(* Logix 5000 project; controller R5_CSS vendor 1 type 14 code 74 rev 19.11; software revision 19.01; part 10 of 20 *)
(* tags used below, declared in another part *)
   CSS_SHUT_PALL : BOOL;
   AlarmMaster : DINT;
   AllowHeatersWhenEmpty : BOOL;
   AllowHeatersWhenEmpty_MaxMin : DINT;
   AllowHeatersWhenEmpty_ONS : BOOL;
   AllowHeatersWhenEmpty_SecRemaining : DINT;
   AllowHeatersWhenEmptyTON : TIMER;
   CSS_Heartbeat : BOOL;
   CSS_HeartbeatTmr : TIMER;
   CSS_HeartbeatToggle : BOOL;
   CSS_OK_TO_RUN : BOOL;   // PRU_RUN_DISABLE 0 = Cannot Run 1 = OK to Run
   CSS_OK_TO_RUN_TOF : TIMER;
   CSS_OK_TO_START : BOOL;   // PRU_START_DISABLE 0 = Cannot Start 1 = OK to Start
   CSS_OK_TO_START_TOF : TIMER;
   HART1 : HARTModuleDef;
   HeaterControl_IgnoreLevel : BOOL;
   HeaterControl_IgnoreLevel_ONS : BOOL;
   LC101 : LEVEL_CONTROL;   // QUENCH TOWER BASIN LIT
   LC205 : LEVEL_CONTROL;   // OVERHEAD CONDENSER BASIN LEVEL CONTROL
   LC205_START_SP : REAL;
   LC205_STOP_SP : REAL;
   LC303A : LEVEL_CONTROL;   // AQUEOUS PHASE OF PRIMARY SETTLER
   LC303B : LEVEL_CONTROL;   // INTERFACE LEVEL OF PRIMARY CONDENSER
   LC303C : LEVEL_CONTROL;   // DIFFERENCE BETWEEN INTERFACE AND AQUEOUS PHASE LT 303
   MV115B : ValveControl_TwoWay;
   MV301 : ValveControl_TwoWay;
   ONE_SHOT : BOOL[32];
   P101A : PUMP_CONTROL;
   P101A_OK : BOOL;
   P101B : PUMP_CONTROL;
   P101B_OK : BOOL;
   P205 : PUMP_CONTROL;   // OVERHEAD CONDENSER TRANSFER PUMP
   P205_QI_AUTO_OS : BOOL;
   P205_QI_MAN_OS : BOOL;
   P302A : PUMP_CONTROL;
   P302A_OK : BOOL;
   P302A_PumpOut : BOOL;
   P302B : PUMP_CONTROL;
   P302B_OK : BOOL;
   P302B_PumpOut : BOOL;
   P303A : PUMP_CONTROL;
   P303A_OK : BOOL;
   P303B : PUMP_CONTROL;
   P303B_OK : BOOL;
   PC407B : PRESSURE_CONTROL;   // POST HX LOW PRESSURE TRANSMITTER
   TC101A : TEMP_CONTROL;   // QUENCH BASIN TRANSFER BASIN A TEMPERATURE CONTROL
   TC101B : TEMP_CONTROL;   // QUENCH BASIN TRANSFER BASIN B TEMPERATURE CONTROL
   TC108 : TEMP_CONTROL;   // QUENCH TOWER EXIT GAS TEMPERATURE CONTROL
   TC112 : TEMP_CONTROL;   // Quench Water Cartridge Heater ProcessTemp
   TC313A : TEMP_CONTROL;   // PRIMARY COALESCER SEPARATOR TEMPERATURE CONTROL
   TC319 : TEMP_CONTROL;   // COALESCER OIL CHAMBER PROCESS TEMPERATURE CONTROL
   TestyBit : DINT;
   TMR_CRIT_FAULT : DINT;
   TMR_FAULT : DINT;
   UTL_Comms : DINT[3];
(* MainProgram, continued *)

ROUTINE LCV303C_COPY_CoalPriChamberInterfaceDiff   (* ladder *)
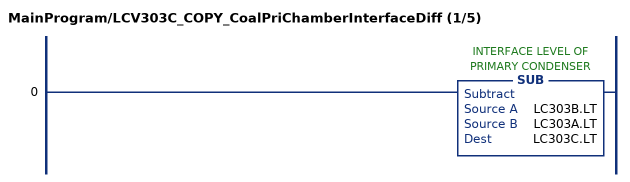
   0: SUB(LC303B.LT,LC303A.LT,LC303C.LT);
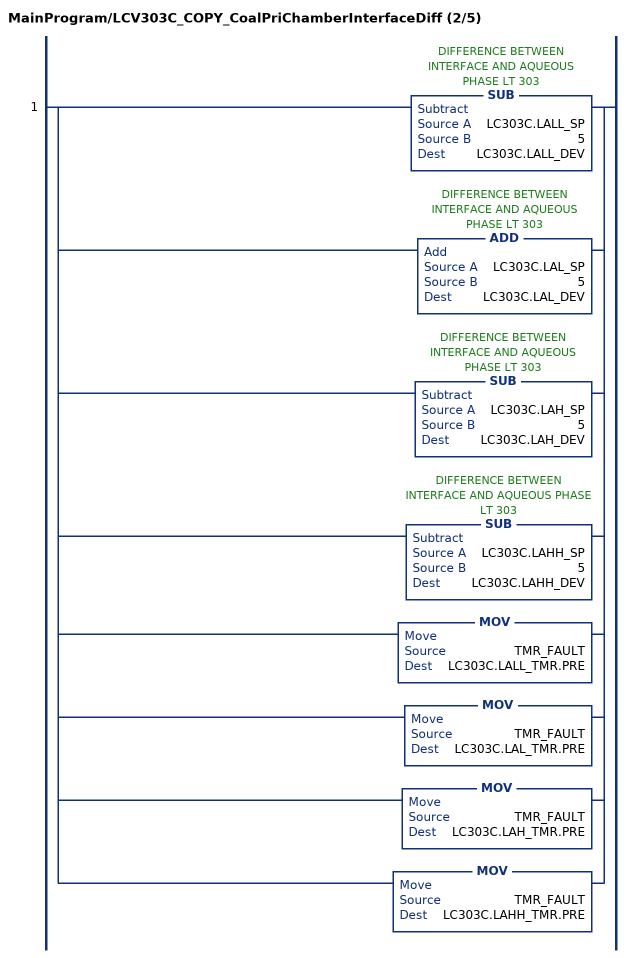
   1: [SUB(LC303C.LALL_SP,5,LC303C.LALL_DEV) ,ADD(LC303C.LAL_SP,5,LC303C.LAL_DEV) ,SUB(LC303C.LAH_SP,5,LC303C.LAH_DEV) ,SUB(LC303C.LAHH_SP,5,LC303C.LAHH_DEV) ,MOV(TMR_FAULT,LC303C.LALL_TMR.PRE) ,MOV(TMR_FAULT,LC303C.LAL_TMR.PRE) ,MOV(TMR_FAULT,LC303C.LAH_TMR.PRE) ,MOV(TMR_FAULT,LC303C.LAHH_TMR.PRE) ];
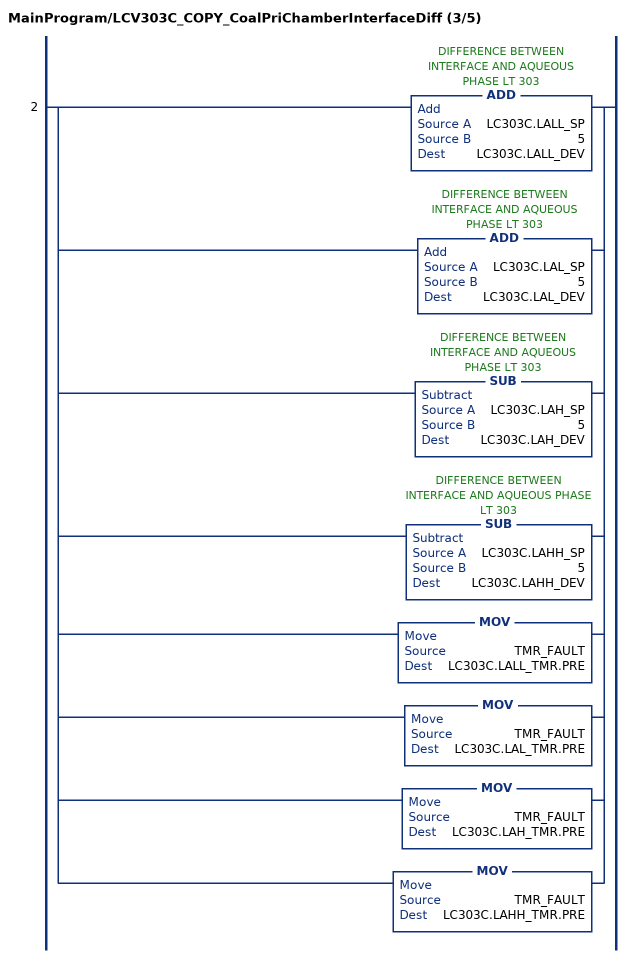
   2: [ADD(LC303C.LALL_SP,5,LC303C.LALL_DEV) ,ADD(LC303C.LAL_SP,5,LC303C.LAL_DEV) ,SUB(LC303C.LAH_SP,5,LC303C.LAH_DEV) ,SUB(LC303C.LAHH_SP,5,LC303C.LAHH_DEV) ,MOV(TMR_FAULT,LC303C.LALL_TMR.PRE) ,MOV(TMR_FAULT,LC303C.LAL_TMR.PRE) ,MOV(TMR_FAULT,LC303C.LAH_TMR.PRE) ,MOV(TMR_FAULT,LC303C.LAHH_TMR.PRE) ];
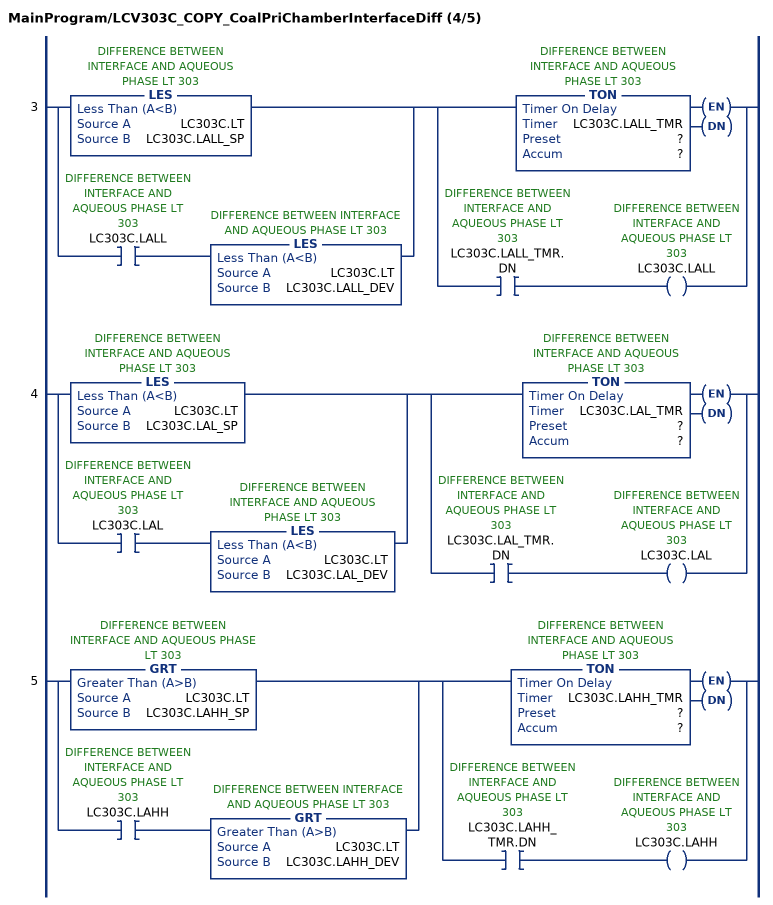
   3: [LES(LC303C.LT,LC303C.LALL_SP) ,XIC(LC303C.LALL) LES(LC303C.LT,LC303C.LALL_DEV) ][TON(LC303C.LALL_TMR,?,?) ,XIC(LC303C.LALL_TMR.DN) OTE(LC303C.LALL) ];
   4: [LES(LC303C.LT,LC303C.LAL_SP) ,XIC(LC303C.LAL) LES(LC303C.LT,LC303C.LAL_DEV) ][TON(LC303C.LAL_TMR,?,?) ,XIC(LC303C.LAL_TMR.DN) OTE(LC303C.LAL) ];
   5: [GRT(LC303C.LT,LC303C.LAHH_SP) ,XIC(LC303C.LAHH) GRT(LC303C.LT,LC303C.LAHH_DEV) ][TON(LC303C.LAHH_TMR,?,?) ,XIC(LC303C.LAHH_TMR.DN) OTE(LC303C.LAHH) ];
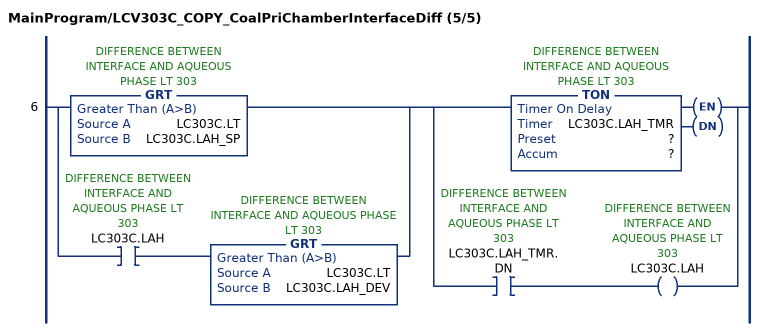
   6: [GRT(LC303C.LT,LC303C.LAH_SP) ,XIC(LC303C.LAH) GRT(LC303C.LT,LC303C.LAH_DEV) ][TON(LC303C.LAH_TMR,?,?) ,XIC(LC303C.LAH_TMR.DN) OTE(LC303C.LAH) ];
END_ROUTINE

ROUTINE MainRoutine   (* ladder *)
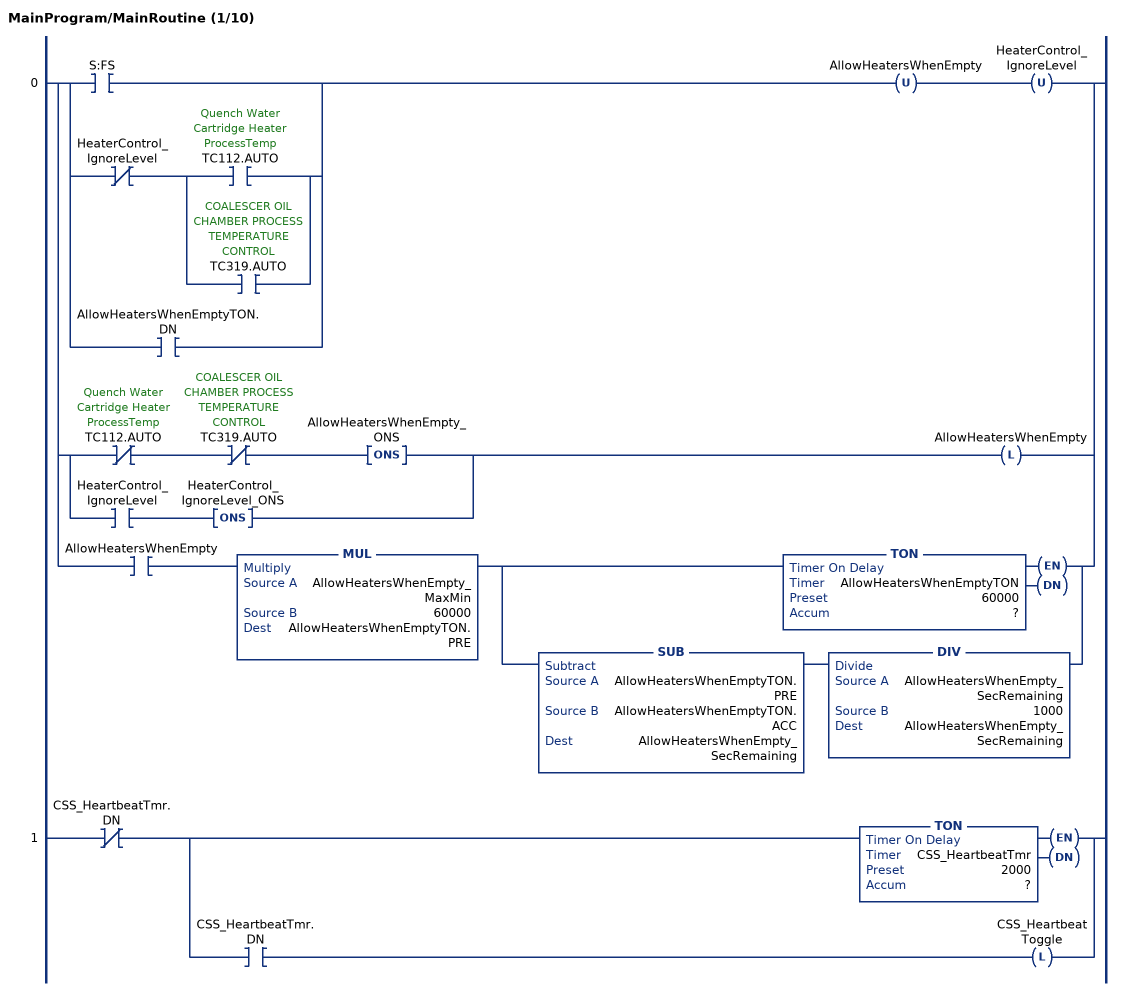
   0: [[XIC(S:FS) ,XIO(HeaterControl_IgnoreLevel) [XIC(TC112.AUTO) ,XIC(TC319.AUTO) ] ,XIC(AllowHeatersWhenEmptyTON.DN) ] OTU(AllowHeatersWhenEmpty) OTU(HeaterControl_IgnoreLevel) ,[XIO(TC112.AUTO) XIO(TC319.AUTO) ONS(AllowHeatersWhenEmpty_ONS) ,XIC(HeaterControl_IgnoreLevel) ONS(HeaterControl_IgnoreLevel_ONS) ] OTL(AllowHeatersWhenEmpty) ,XIC(AllowHeatersWhenEmpty) MUL(AllowHeatersWhenEmpty_MaxMin,60000,AllowHeatersWhenEmptyTON.PRE) [TON(AllowHeatersWhenEmptyTON,?,?) ,SUB(AllowHeatersWhenEmptyTON.PRE,AllowHeatersWhenEmptyTON.ACC,AllowHeatersWhenEmpty_SecRemaining) DIV(AllowHeatersWhenEmpty_SecRemaining,1000,AllowHeatersWhenEmpty_SecRemaining) ] ];
   1: XIO(CSS_HeartbeatTmr.DN)[TON(CSS_HeartbeatTmr,?,?) ,XIC(CSS_HeartbeatTmr.DN) OTL(CSS_HeartbeatToggle) ];
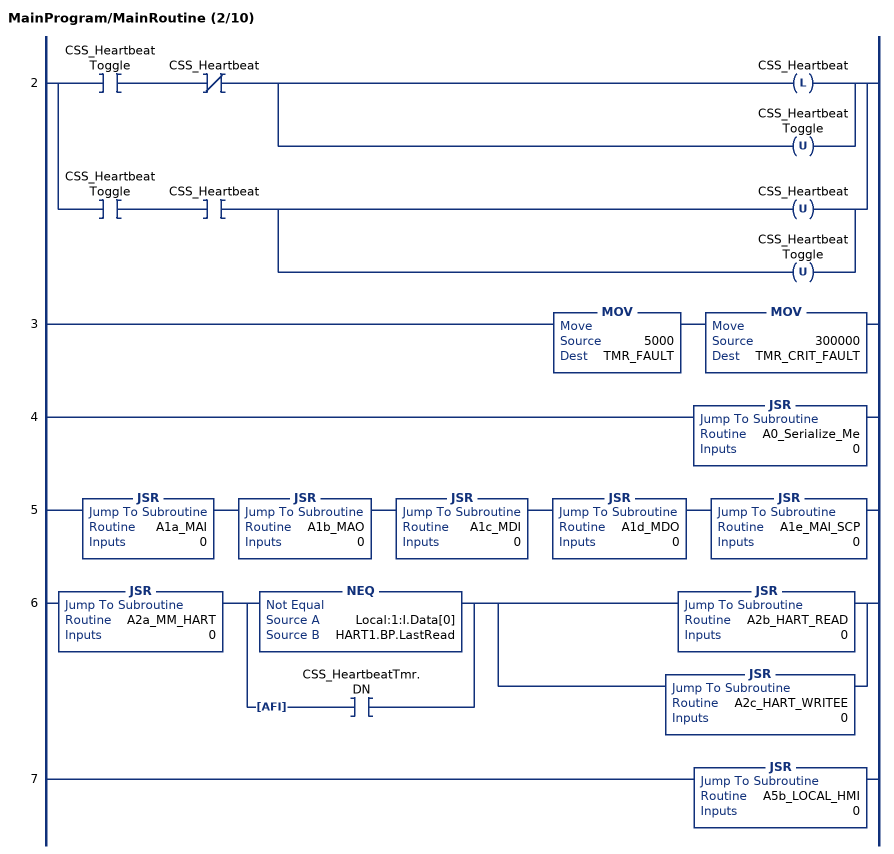
   2: [XIC(CSS_HeartbeatToggle) XIO(CSS_Heartbeat) [OTL(CSS_Heartbeat) ,OTU(CSS_HeartbeatToggle) ] ,XIC(CSS_HeartbeatToggle) XIC(CSS_Heartbeat) [OTU(CSS_Heartbeat) ,OTU(CSS_HeartbeatToggle) ] ];
   3: MOV(5000,TMR_FAULT)MOV(300000,TMR_CRIT_FAULT);
   4: JSR(A0_Serialize_Me,0);
   5: JSR(A1a_MAI,0)JSR(A1b_MAO,0)JSR(A1c_MDI,0)JSR(A1d_MDO,0)JSR(A1e_MAI_SCP,0);
   6: JSR(A2a_MM_HART,0)[NEQ(Local:1:I.Data[0],HART1.BP.LastRead) ,AFI() XIC(CSS_HeartbeatTmr.DN) ][JSR(A2b_HART_READ,0) ,JSR(A2c_HART_WRITEE,0) ];
   7: JSR(A5b_LOCAL_HMI,0);
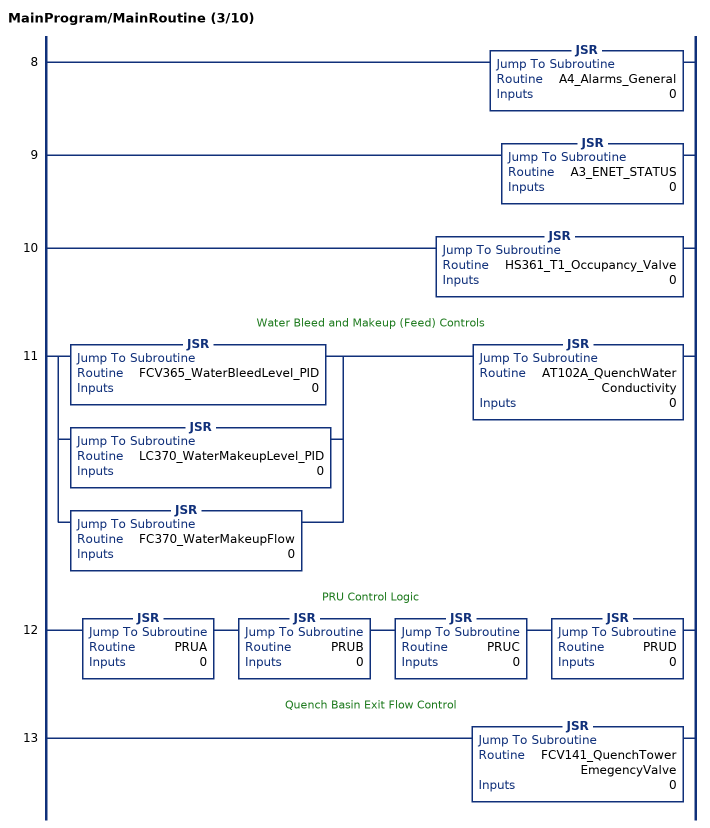
   8: JSR(A4_Alarms_General,0);
   9: JSR(A3_ENET_STATUS,0);
   10: JSR(HS361_T1_Occupancy_Valve,0);
   // Water Bleed and Makeup (Feed) Controls
   11: [JSR(FCV365_WaterBleedLevel_PID,0) ,JSR(LC370_WaterMakeupLevel_PID,0) ,JSR(FC370_WaterMakeupFlow,0) ]JSR(AT102A_QuenchWaterConductivity,0);
   // PRU Control Logic
   12: JSR(PRUA,0)JSR(PRUB,0)JSR(PRUC,0)JSR(PRUD,0);
   // Quench Basin Exit Flow Control
   13: JSR(FCV141_QuenchTowerEmegencyValve,0);
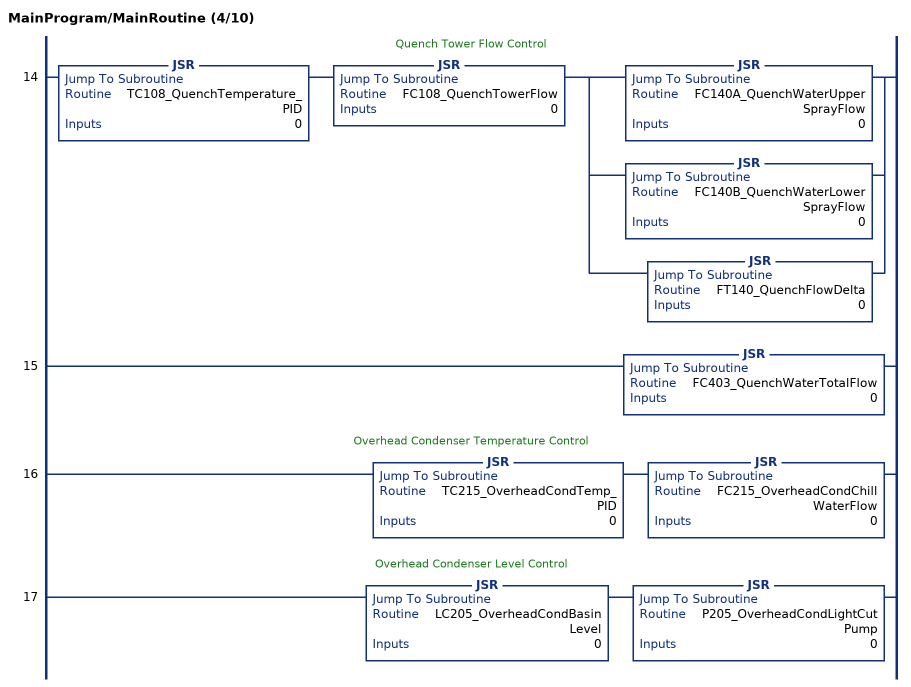
   // Quench Tower Flow Control
   14: JSR(TC108_QuenchTemperature_PID,0)JSR(FC108_QuenchTowerFlow,0)[JSR(FC140A_QuenchWaterUpperSprayFlow,0) ,JSR(FC140B_QuenchWaterLowerSprayFlow,0) ,JSR(FT140_QuenchFlowDelta,0) ];
   15: JSR(FC403_QuenchWaterTotalFlow,0);
   // Overhead Condenser Temperature Control
   16: JSR(TC215_OverheadCondTemp_PID,0)JSR(FC215_OverheadCondChillWaterFlow,0);
   // Overhead Condenser Level Control
   17: JSR(LC205_OverheadCondBasinLevel,0)JSR(P205_OverheadCondLightCutPump,0);
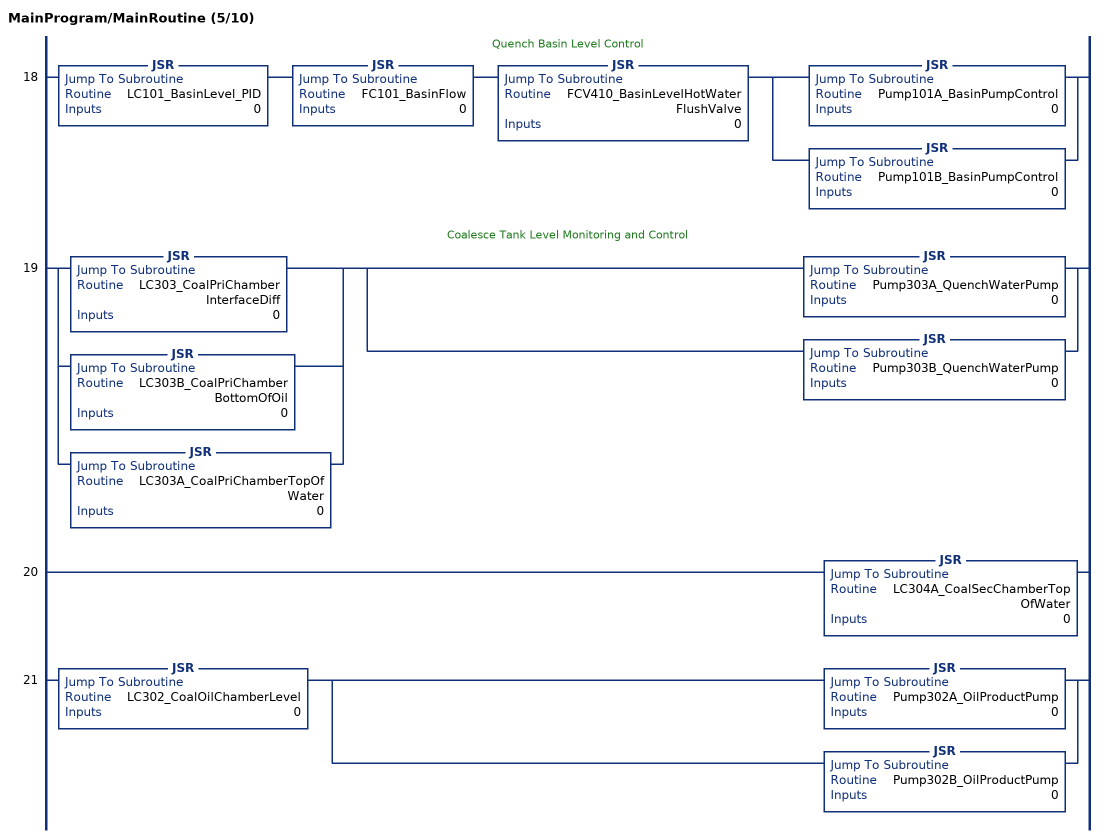
   // Quench Basin Level Control
   18: JSR(LC101_BasinLevel_PID,0)JSR(FC101_BasinFlow,0)JSR(FCV410_BasinLevelHotWaterFlushValve,0)[JSR(Pump101A_BasinPumpControl,0) ,JSR(Pump101B_BasinPumpControl,0) ];
   // Coalesce Tank Level Monitoring and Control
   19: [JSR(LC303_CoalPriChamberInterfaceDiff,0) ,JSR(LC303B_CoalPriChamberBottomOfOil,0) ,JSR(LC303A_CoalPriChamberTopOfWater,0) ][JSR(Pump303A_QuenchWaterPump,0) ,JSR(Pump303B_QuenchWaterPump,0) ];
   20: JSR(LC304A_CoalSecChamberTopOfWater,0);
   21: JSR(LC302_CoalOilChamberLevel,0)[JSR(Pump302A_OilProductPump,0) ,JSR(Pump302B_OilProductPump,0) ];
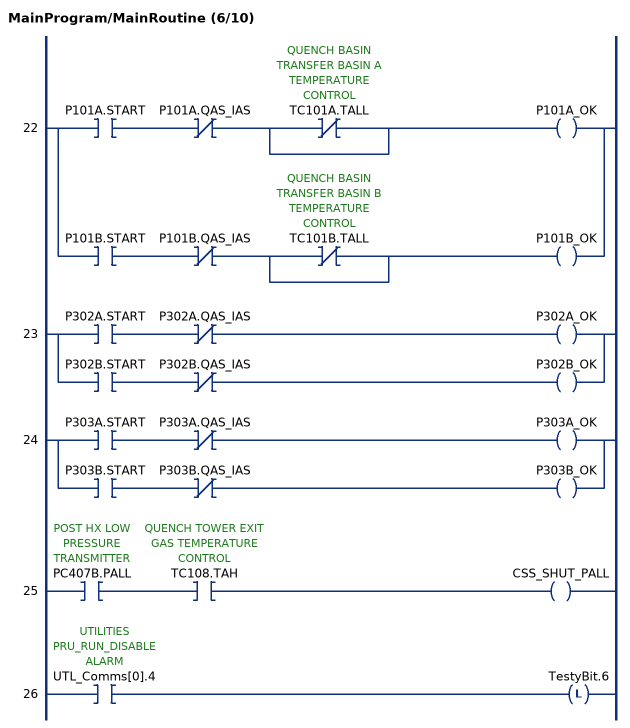
   22: [XIC(P101A.START) XIO(P101A.QAS_IAS) [XIO(TC101A.TALL) ,] OTE(P101A_OK) ,XIC(P101B.START) XIO(P101B.QAS_IAS) [XIO(TC101B.TALL) ,] OTE(P101B_OK) ];
   23: [XIC(P302A.START) XIO(P302A.QAS_IAS) OTE(P302A_OK) ,XIC(P302B.START) XIO(P302B.QAS_IAS) OTE(P302B_OK) ];
   24: [XIC(P303A.START) XIO(P303A.QAS_IAS) OTE(P303A_OK) ,XIC(P303B.START) XIO(P303B.QAS_IAS) OTE(P303B_OK) ];
   25: XIC(PC407B.PALL)XIC(TC108.TAH)OTE(CSS_SHUT_PALL);
   26: XIC(UTL_Comms[0].4)OTL(TestyBit.6);
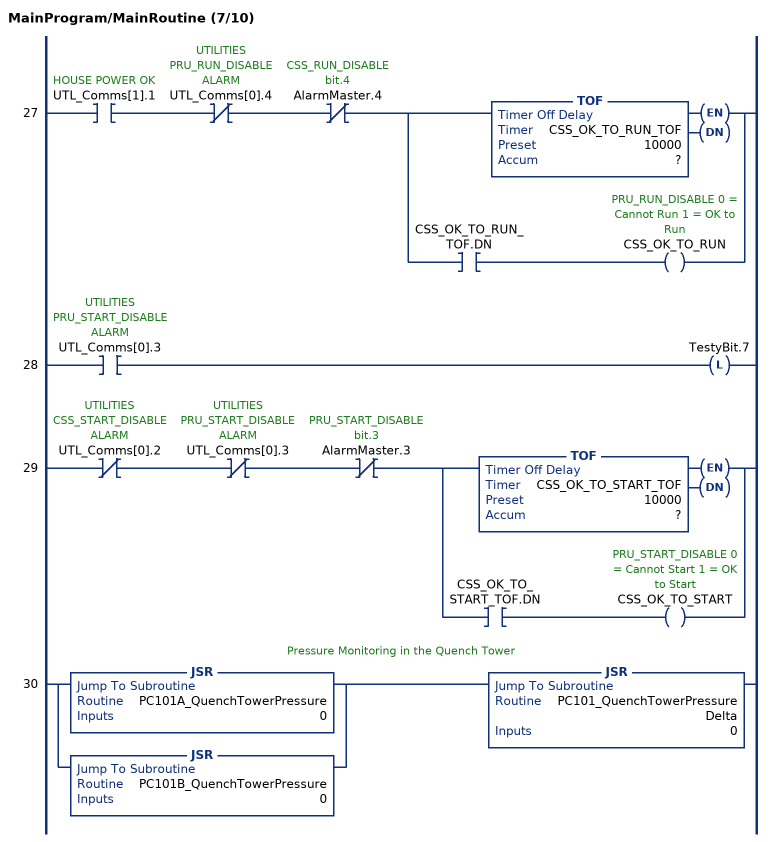
   27: XIC(UTL_Comms[1].1)XIO(UTL_Comms[0].4)XIO(AlarmMaster.4)[TOF(CSS_OK_TO_RUN_TOF,?,?) ,XIC(CSS_OK_TO_RUN_TOF.DN) OTE(CSS_OK_TO_RUN) ];
   28: XIC(UTL_Comms[0].3)OTL(TestyBit.7);
   29: XIO(UTL_Comms[0].2)XIO(UTL_Comms[0].3)XIO(AlarmMaster.3)[TOF(CSS_OK_TO_START_TOF,?,?) ,XIC(CSS_OK_TO_START_TOF.DN) OTE(CSS_OK_TO_START) ];
   // Pressure Monitoring in the Quench Tower
   30: [JSR(PC101A_QuenchTowerPressure,0) ,JSR(PC101B_QuenchTowerPressure,0) ]JSR(PC101_QuenchTowerPressureDelta,0);
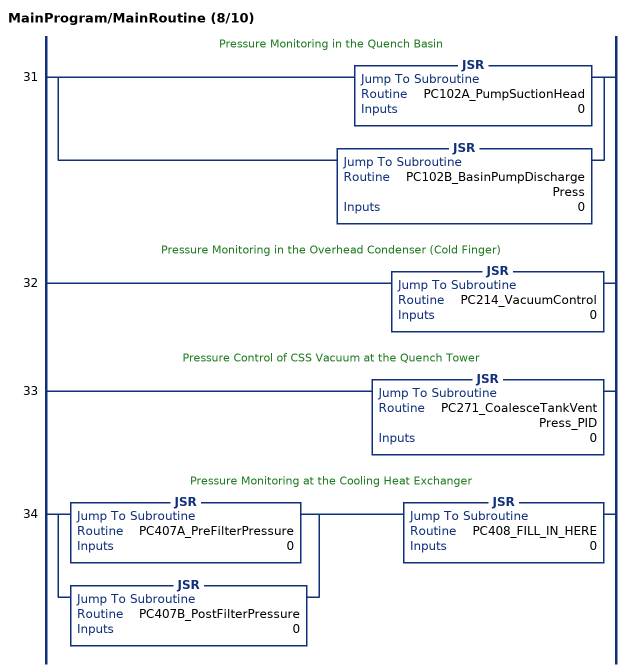
   // Pressure Monitoring in the Quench Basin
   31: [JSR(PC102A_PumpSuctionHead,0) ,JSR(PC102B_BasinPumpDischargePress,0) ];
   // Pressure Monitoring in the Overhead Condenser (Cold Finger)
   32: JSR(PC214_VacuumControl,0);
   // Pressure Control of CSS Vacuum at the Quench Tower
   33: JSR(PC271_CoalesceTankVentPress_PID,0);
   // Pressure Monitoring at the Cooling Heat Exchanger
   34: [JSR(PC407A_PreFilterPressure,0) ,JSR(PC407B_PostFilterPressure,0) ]JSR(PC408_FILL_IN_HERE,0);
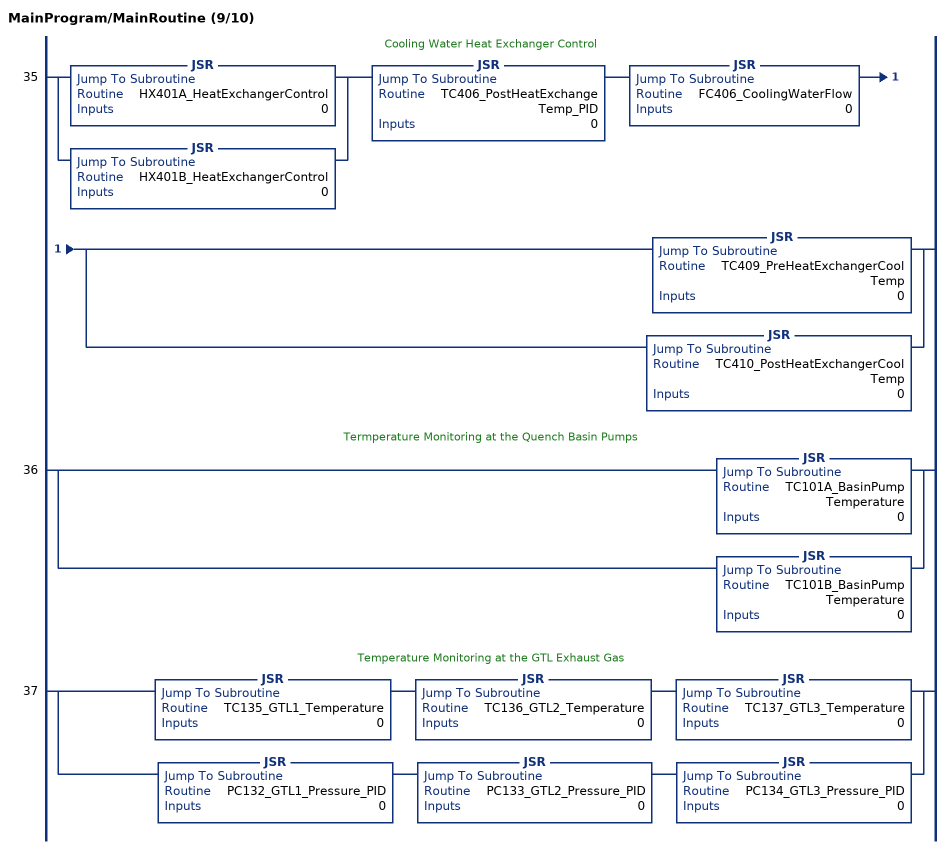
   // Cooling Water Heat Exchanger Control
   35: [JSR(HX401A_HeatExchangerControl,0) ,JSR(HX401B_HeatExchangerControl,0) ]JSR(TC406_PostHeatExchangeTemp_PID,0)JSR(FC406_CoolingWaterFlow,0)[JSR(TC409_PreHeatExchangerCoolTemp,0) ,JSR(TC410_PostHeatExchangerCoolTemp,0) ];
   // Termperature Monitoring at the Quench Basin Pumps
   36: [JSR(TC101A_BasinPumpTemperature,0) ,JSR(TC101B_BasinPumpTemperature,0) ];
   // Temperature Monitoring at the GTL Exhaust Gas
   37: [JSR(TC135_GTL1_Temperature,0) JSR(TC136_GTL2_Temperature,0) JSR(TC137_GTL3_Temperature,0) ,JSR(PC132_GTL1_Pressure_PID,0) JSR(PC133_GTL2_Pressure_PID,0) JSR(PC134_GTL3_Pressure_PID,0) ];
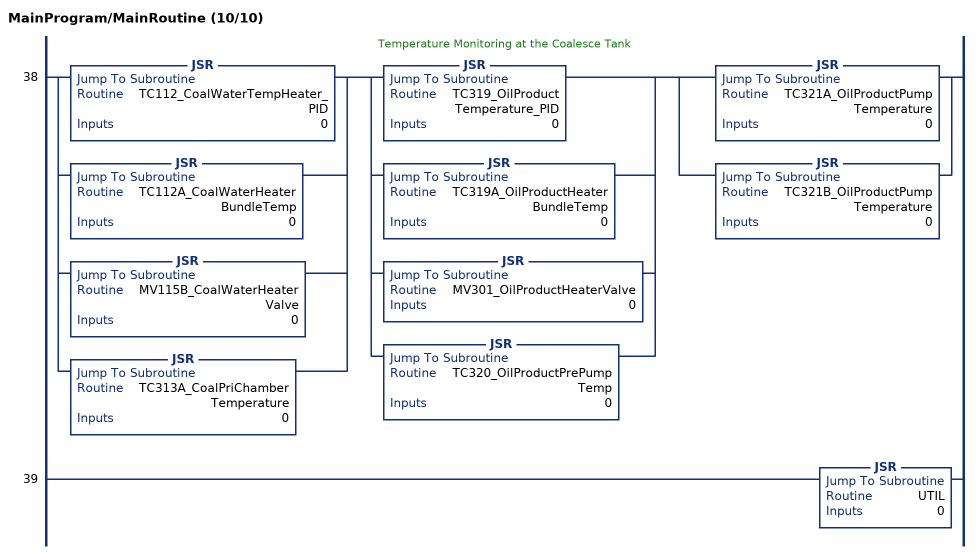
   // Temperature Monitoring at the Coalesce Tank
   38: [JSR(TC112_CoalWaterTempHeater_PID,0) ,JSR(TC112A_CoalWaterHeaterBundleTemp,0) ,JSR(MV115B_CoalWaterHeaterValve,0) ,JSR(TC313A_CoalPriChamberTemperature,0) ][JSR(TC319_OilProductTemperature_PID,0) ,JSR(TC319A_OilProductHeaterBundleTemp,0) ,JSR(MV301_OilProductHeaterValve,0) ,JSR(TC320_OilProductPrePumpTemp,0) ][JSR(TC321A_OilProductPumpTemperature,0) ,JSR(TC321B_OilProductPumpTemperature,0) ];
   39: JSR(UTIL,0);
END_ROUTINE

ROUTINE MV115B_CoalWaterHeaterValve   (* ladder *)
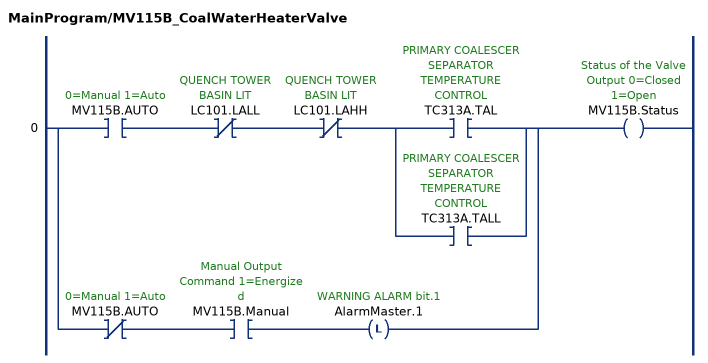
   0: [XIC(MV115B.AUTO) XIO(LC101.LALL) XIO(LC101.LAHH) [XIC(TC313A.TAL) ,XIC(TC313A.TALL) ] ,XIO(MV115B.AUTO) XIC(MV115B.Manual) OTL(AlarmMaster.1) ]OTE(MV115B.Status);
END_ROUTINE

ROUTINE MV301_OilProductHeaterValve   (* ladder *)
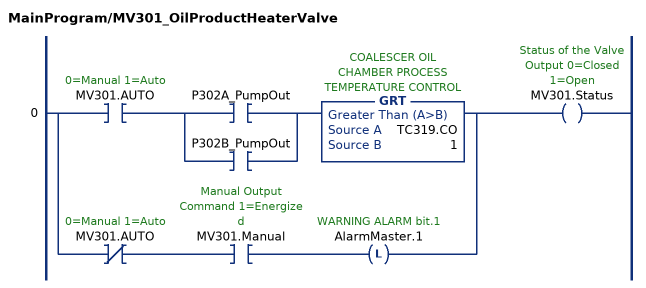
   0: [XIC(MV301.AUTO) [XIC(P302A_PumpOut) ,XIC(P302B_PumpOut) ] GRT(TC319.CO,1) ,XIO(MV301.AUTO) XIC(MV301.Manual) OTL(AlarmMaster.1) ]OTE(MV301.Status);
END_ROUTINE

ROUTINE P205_OverheadCondLightCutPump   (* ladder *)
// OVERHEAD CONDENSER
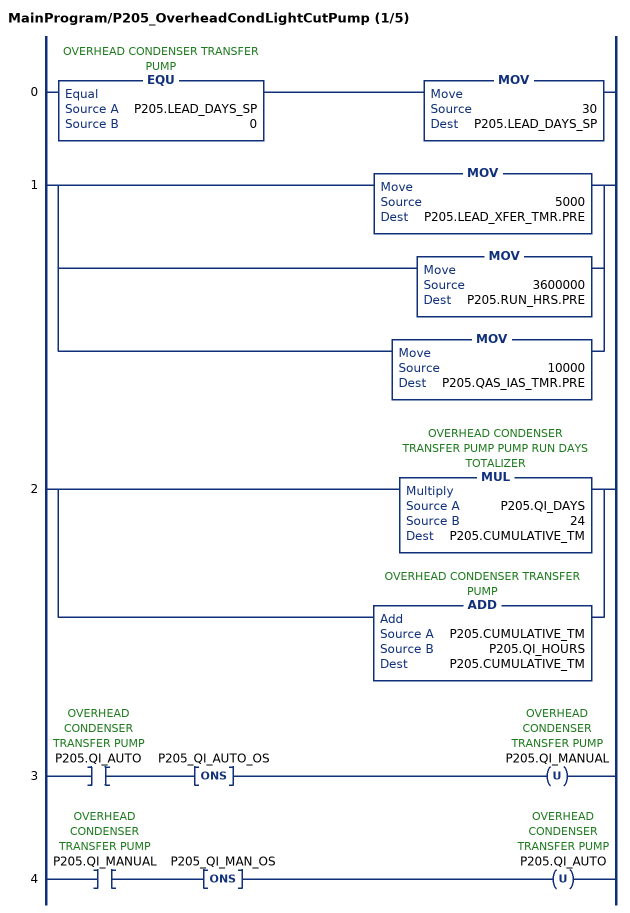
   0: EQU(P205.LEAD_DAYS_SP,0)MOV(30,P205.LEAD_DAYS_SP);
   1: [MOV(5000,P205.LEAD_XFER_TMR.PRE) ,MOV(3600000,P205.RUN_HRS.PRE) ,MOV(10000,P205.QAS_IAS_TMR.PRE) ];
   2: [MUL(P205.QI_DAYS,24,P205.CUMULATIVE_TM) ,ADD(P205.CUMULATIVE_TM,P205.QI_HOURS,P205.CUMULATIVE_TM) ];
   3: XIC(P205.QI_AUTO)ONS(P205_QI_AUTO_OS)OTU(P205.QI_MANUAL);
   4: XIC(P205.QI_MANUAL)ONS(P205_QI_MAN_OS)OTU(P205.QI_AUTO);
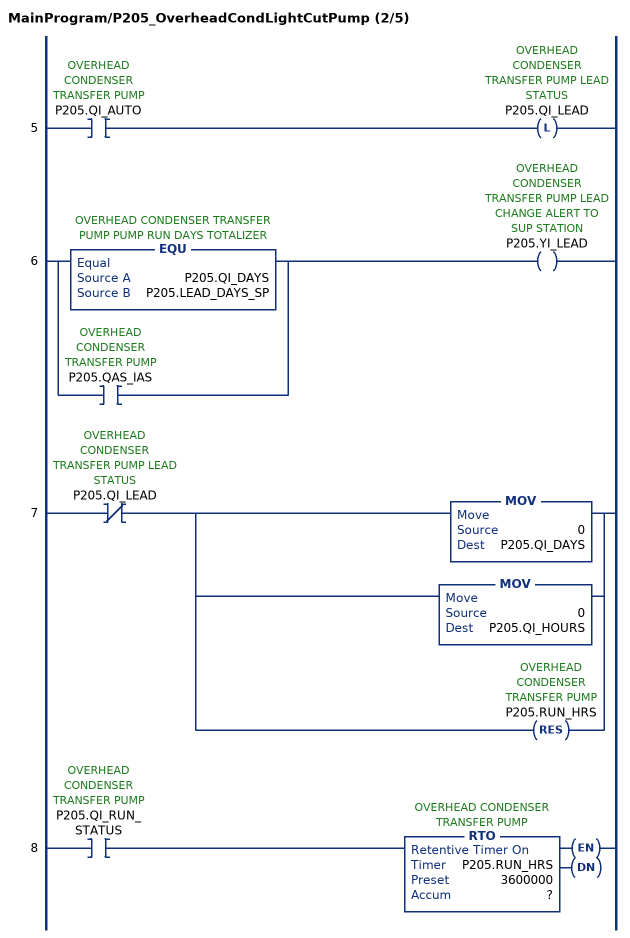
   5: XIC(P205.QI_AUTO)OTL(P205.QI_LEAD);
   6: [EQU(P205.QI_DAYS,P205.LEAD_DAYS_SP) ,XIC(P205.QAS_IAS) ]OTE(P205.YI_LEAD);
   7: XIO(P205.QI_LEAD)[MOV(0,P205.QI_DAYS) ,MOV(0,P205.QI_HOURS) ,RES(P205.RUN_HRS) ];
   8: XIC(P205.QI_RUN_STATUS)RTO(P205.RUN_HRS,?,?);
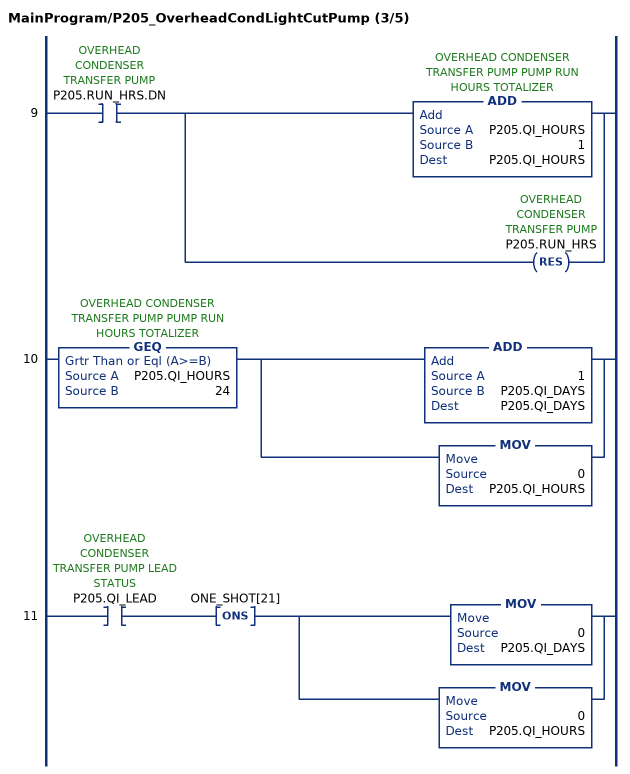
   9: XIC(P205.RUN_HRS.DN)[ADD(P205.QI_HOURS,1,P205.QI_HOURS) ,RES(P205.RUN_HRS) ];
   10: GEQ(P205.QI_HOURS,24)[ADD(1,P205.QI_DAYS,P205.QI_DAYS) ,MOV(0,P205.QI_HOURS) ];
   11: XIC(P205.QI_LEAD)ONS(ONE_SHOT[21])[MOV(0,P205.QI_DAYS) ,MOV(0,P205.QI_HOURS) ];
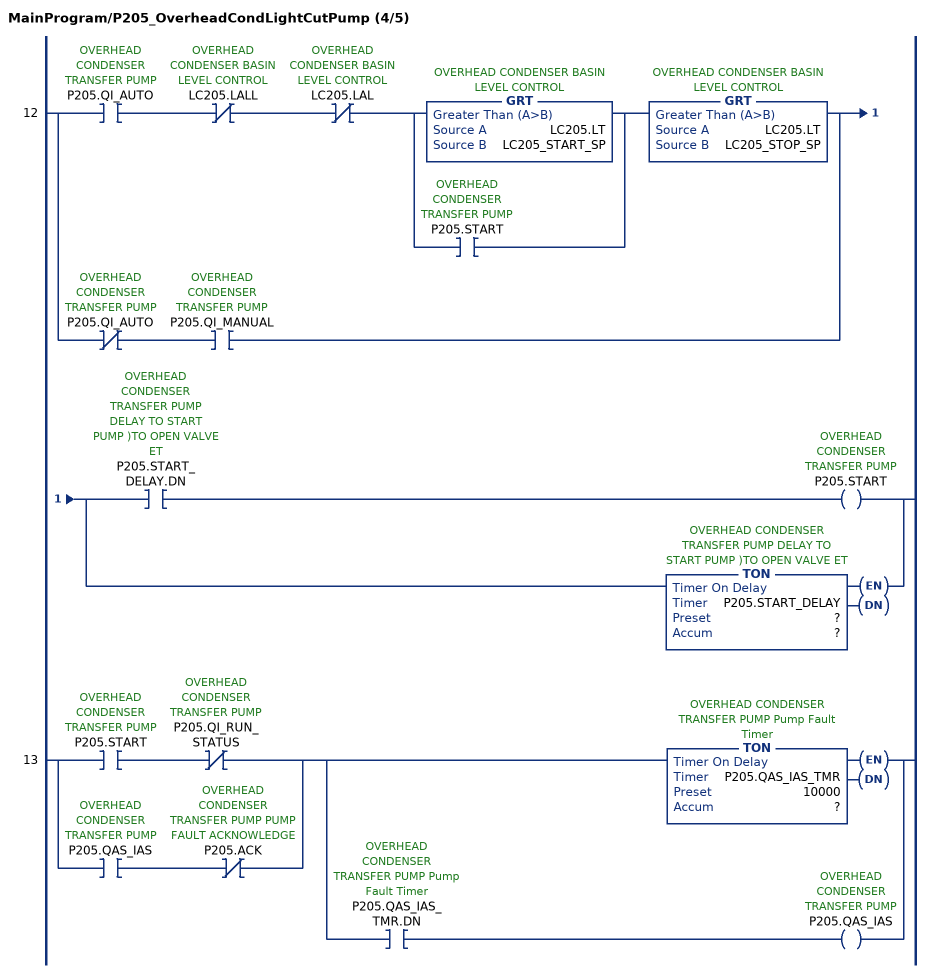
   12: [XIC(P205.QI_AUTO) XIO(LC205.LALL) XIO(LC205.LAL) [GRT(LC205.LT,LC205_START_SP) ,XIC(P205.START) ] GRT(LC205.LT,LC205_STOP_SP) ,XIO(P205.QI_AUTO) XIC(P205.QI_MANUAL) ][XIC(P205.START_DELAY.DN) OTE(P205.START) ,TON(P205.START_DELAY,?,?) ];
   13: [XIC(P205.START) XIO(P205.QI_RUN_STATUS) ,XIC(P205.QAS_IAS) XIO(P205.ACK) ][TON(P205.QAS_IAS_TMR,?,?) ,XIC(P205.QAS_IAS_TMR.DN) OTE(P205.QAS_IAS) ];
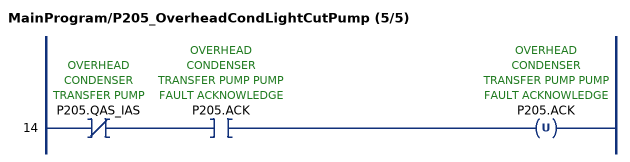
   14: XIO(P205.QAS_IAS)XIC(P205.ACK)OTU(P205.ACK);
END_ROUTINE
